FUNCTION_BLOCK FB_Flender_DamageReader
VAR_INPUT
	TimeOffset 		: T_MAXSTRING; 
	ReadInterval 	: TIME := T#1M; 
	Ip				: T_IPv4Addr := '127.0.0.1'; 
	
END_VAR
VAR
	iTest 	: UDINT; 
	
	Timer : TON; 
	bRead : BOOL; 
	
	Tags 	: ARRAY[0..50] OF T_MAXSTRING;
	Values 	: ARRAY[0..50] OF LREAL; 
	
	reader	: FB_InfluxReader; 
	CurrentState : 	E_InfluxReaderState;
END_VAR
VAR_IN_OUT
	Dmg_Foundation 	: LREAL;
	Dmg_Footplates 	: LREAL;
	Dmg_MBS			: LREAL;	
	Dmg_LU1			: LREAL; 
	Dmg_LU2			: LREAL; 
END_VAR

iTest := iTest + 1;

Timer( 	IN 	:= NOT(Timer.Q),
		PT 	:= ReadInterval,
		Q	=> bRead); 

IF bRead THEN
	bRead := FALSE;
	reader.ReadValues();
END_IF
// ========= Setup Values
	Tags[0] := 'General_Foundation_Lu1';
	Tags[1] := 'General_Foundation_Lu2';
	
	Tags[2] := 'General_Footplates_Lu1';
	Tags[3] := 'General_Footplates_Lu2';
	
	Tags[4] := 'General_MBS_Lu1';
	Tags[5] := 'General_MBS_Lu2';
	
	Tags[6] := 'General_Platform_Lu1';
	Tags[7] := 'General_Platform_Lu2';

// ======== Run Reader
	reader(	Ip					:= Ip, 
			Port				:= 8086, 
			ReplyReadInterval	:= T#200MS, 
			InfluxDatabase		:= 'RD_Damage', 
			InfluxMeasurement	:= 'DamageCalculation', 
			ValuesToFind		:= 8, 
			ValueNames			:= Tags,
			TimeOffset			:= TimeOffset,
			ValuesRead			=> Values,
			CurrentState		=> CurrentState);
		
		
// ======= Output Values
	Dmg_Foundation 	:= UpdateCurrentValue(Dmg_Foundation, Values[0], Values[1]);
	Dmg_Footplates 	:= UpdateCurrentValue(Dmg_Footplates, Values[2], Values[3]);
	Dmg_MBS			:= UpdateCurrentValue(Dmg_MBS, Values[4], Values[5]); 
	Dmg_LU1			:= UpdateCurrentValue(Dmg_LU1, Values[6], 0);
	Dmg_LU2			:= UpdateCurrentValue(Dmg_LU1, Values[7], 0);

METHOD PRIVATE UpdateCurrentValue : LREAL
VAR_INPUT
	CurrentValue : LREAL;
	Lu1Value	: LREAL;
	Lu2Value 	: LREAL; 
END_VAR
VAR
	newestMaxValue : LREAL; 
	outputValue : LREAL;
END_VAR


newestMaxValue := MAX(Lu1Value, Lu2Value);


outputValue := MAX(CurrentValue, newestMaxValue); 

UpdateCurrentValue := outputValue;
END_METHOD

END_FUNCTION_BLOCK

(* stored: Version 1.1.0.1, ProductVersion 3.1.4022.11
   POU FB_Flender_DamageReader: Id {7ffb4158-7733-41f2-87da-51bcad9e2179}, SpecialFunc None
   Method UpdateCurrentValue: Id {f14b5143-d7f5-4427-b156-9f717fbd18e4} *)
